Fanuc KAREL source: kb00099.KL

PROGRAM KB00099
%STACKSIZE=65535
%PRIORITY=65535
%NOLOCKGROUP
VAR
P1 : STRING[80]
P2 : STRING[80]
RESULT : INTEGER
BEGIN
P1='A'
P2='A'
-- UNRESOLVED_PC line 10 opcodes [27 22 2A 22 2A 76 23] marker_code=28
END KB00099
